// TIA Portal V16 export
// export: Created 2022-03-06T01:32:52.2168537Z, ExportSetting WithDefaults, DisplayName Totally Integrated Automation Portal, DisplayVersion V16 Update 4, DisplayName TIA Portal Version Control Interface, DisplayVersion V16 Update 2, DisplayName TIA Portal Openness, DisplayVersion V16 Update 4, DisplayName TIA Portal Teamcenter Gateway, DisplayVersion V16, DisplayName SINAMICS Startdrive Advanced, DisplayVersion V16 Update 4, DisplayName SINAMICS Startdrive G110M, G120, G120C, G120D, G120P, G115D, DisplayVersion V16 Update 4, DisplayName SINAMICS Startdrive G130, G150, S120, S150, SINAMICS MV, S210, DisplayVersion V16 Update 4, DisplayName STEP 7 Professional, DisplayVersion V16 Update 4, DisplayName STEP 7 Safety, DisplayVersion V16, DisplayName WinCC Advanced / Unified PC, DisplayVersion V16 Update 4
FUNCTION "Linea1" : Void   // FC2, LAD
{ S7_Optimized_Access := 'TRUE' }
VERSION : 0.1
// stored: AutoNumber true, IsIECCheckEnabled false, SetENOAutomatically false, UDAEnableTagReadback false
BEGIN

REGION Network 1
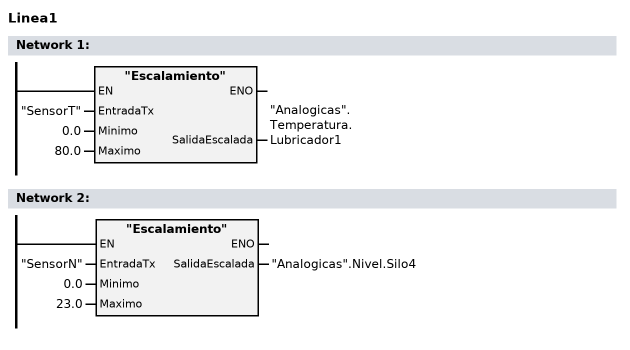
   RUNG wire#powerrail
      "Escalamiento"(EntradaTx := "SensorT", Minimo := 0.0, Maximo := 80.0, SalidaEscalada => "Analogicas".Temperatura.Lubricador1)
   END_RUNG
   // the same network as SCL:
   "Escalamiento"(EntradaTx := "SensorT",
                  Minimo := 0.0,
                  Maximo := 80.0,
                  SalidaEscalada => "Analogicas".Temperatura.Lubricador1);
END_REGION

REGION Network 2
   RUNG wire#powerrail
      "Escalamiento"(EntradaTx := "SensorN", Minimo := 0.0, Maximo := 23.0, SalidaEscalada => "Analogicas".Nivel.Silo4)
   END_RUNG
   // the same network as SCL:
   "Escalamiento"(EntradaTx := "SensorN",
                  Minimo := 0.0,
                  Maximo := 23.0,
                  SalidaEscalada => "Analogicas".Nivel.Silo4);
END_REGION
END_FUNCTION
